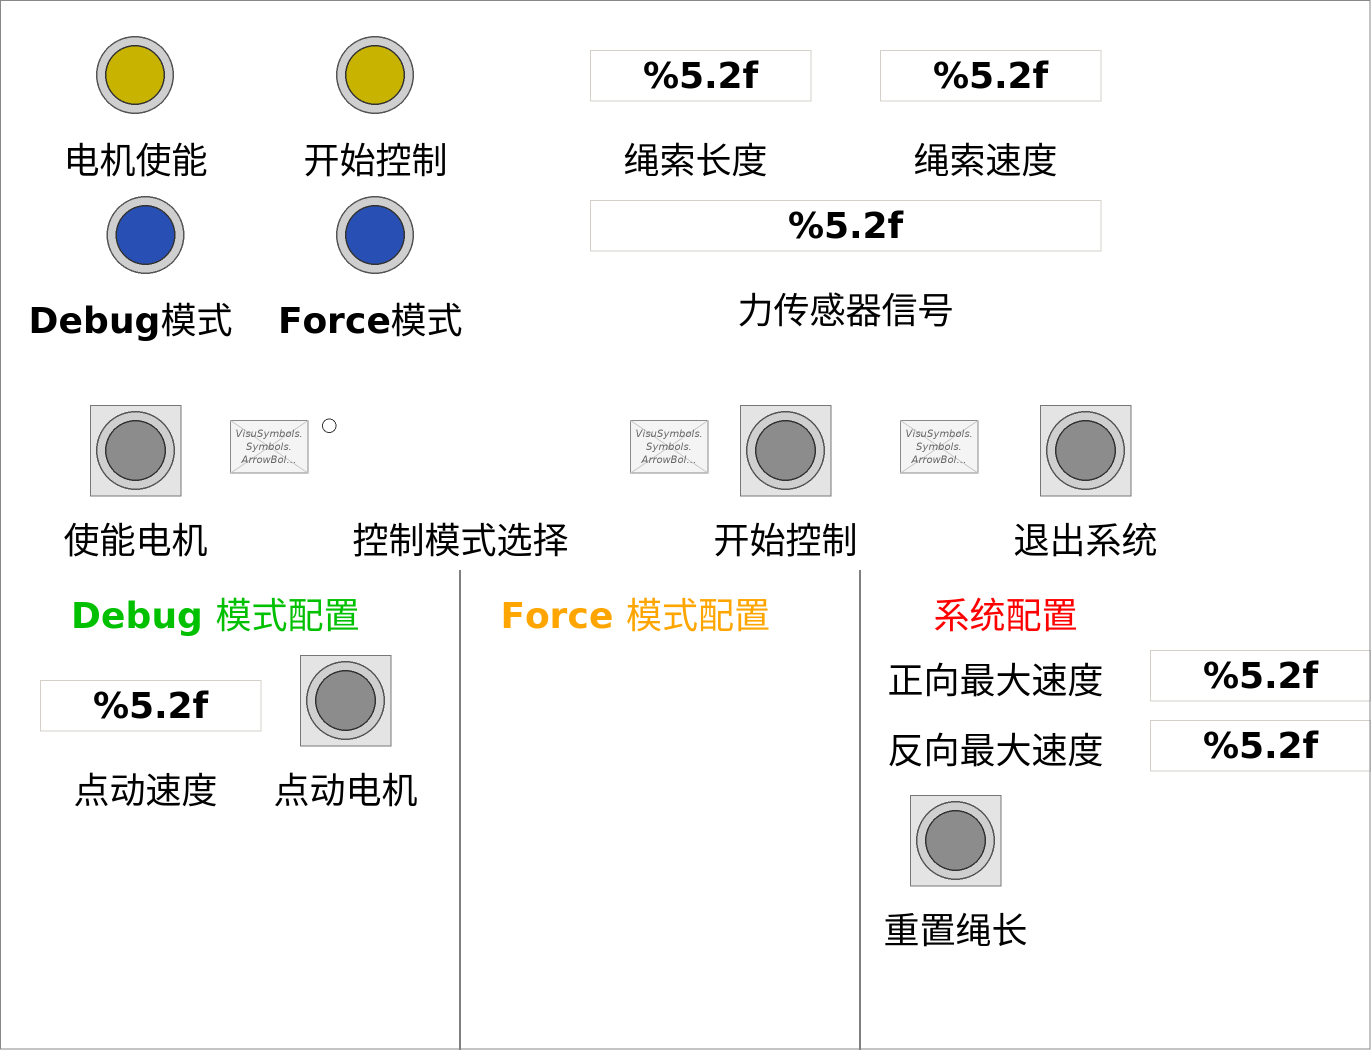
VISUALIZATION ControlHMI  // 1371x1050
    Lamp1 (90,30 90x90), variable: Main.motor_state.is_motor_closedloop, style: Lamp-Lamp1-Yellow
    Label (40,130 191x61), "电机使能"
    Lamp1 (330,30 90x90), variable: Main.system_control_param.is_system_control, style: Lamp-Lamp1-Yellow
    Label (280,130 191x61), "开始控制"
    Label (20,290 221x61), "Debug模式"
    Lamp1 (100,190 91x90), variable: Main.system_control_param.system_control_mode=SystemControlMode.Debug, style: Lamp-Lamp1-Blue
    Label (260,290 221x61), "Force模式"
    Lamp1 (330,190 90x90), variable: Main.system_control_param.system_control_mode=SystemControlMode.ConstForce, style: Lamp-Lamp1-Blue
    Textfield (590,50 221x51), "%5.2f", text variable: Main.motor_state.cable_position
    Label (600,130 191x61), "绳索长度"
    Label (890,130 191x61), "绳索速度"
    Textfield (880,50 221x51), "%5.2f", text variable: Main.motor_state.cable_velocity
    Label (600,280 491x61), "力传感器信号"
    Textfield (590,200 511x51), "%5.2f", text variable: Main.sensor_data.force_value_raw
    PushSwitchLed (90,400 91x101), variable: Main.system_control_param.is_motor_poweron, behaviour: TAP, style: Switch-PushSwitchLed-Gray
    Label (40,510 191x61), "使能电机"
    Image (230,420 78x53), image: VisuSymbols.Symbols.ArrowBoldRight
    RadioButton (320,340 301x171), variable: Main.system_control_param.system_control_mode
        Areas[0]: Text=Debug
        Areas[1]: Text=ConstForce
    Label (310,510 301x61), "控制模式选择"
    Image (630,420 78x53), image: VisuSymbols.Symbols.ArrowBoldRight
    PushSwitchLed (740,400 91x101), variable: Main.system_control_param.is_system_control, behaviour: TOGGLE, style: Switch-PushSwitchLed-Gray
    Label (690,510 191x61), "开始控制"
    Line (460,1050) (460,570)
    PushSwitchLed (1040,400 91x101), variable: Main.system_control_param.is_system_exit, behaviour: TOGGLE, style: Switch-PushSwitchLed-Gray
    Label (990,510 191x61), "退出系统"
    Image (900,420 78x53), image: VisuSymbols.Symbols.ArrowBoldRight
    Label (40,580 351x71), "Debug 模式配置"
    Label (250,760 191x61), "点动电机"
    PushSwitchLed (300,650 91x101), variable: Main.system_control_param.is_motor_jog, behaviour: TAP, style: Switch-PushSwitchLed-Gray
    Textfield (40,680 221x51), "%5.2f", text variable: Main.system_control_param.jog_param.jog_velocity
        OnMouseClick: write the text variable via Default
    Label (50,760 191x61), "点动速度"
    Label (460,580 351x71), "Force 模式配置"
    Line (860,1050) (860,570)
    Label (830,580 351x71), "系统配置"
    Textfield (1150,650 221x51), "%5.2f", text variable: Main.motor_param.max_cable_velocity
        OnMouseClick: write the text variable via Default
    Label (860,650 271x61), "正向最大速度"
    Label (860,720 271x61), "反向最大速度"
    Textfield (1150,720 221x51), "%5.2f", text variable: Main.motor_param.min_cable_velocity
        OnMouseClick: write the text variable via Default
    PushSwitchLed (910,790 91x101), variable: Main.system_control_param.motor_degree2cable_position_param.reset_cable_position, behaviour: TAP, style: Switch-PushSwitchLed-Gray
    Label (860,900 191x61), "重置绳长"
END_VISUALIZATION

(* stored: Version 1.1.0.1, ProductVersion 3.1.4024.11
   Visu ControlHMI: Id {b806a2e9-bf0f-4095-8af3-27bd3dcc66e0} *)
